Fanuc KAREL source: test_lam.kl

PROGRAM test_lam
%NOLOCKGROUP

%include lam.klt

%include default_lam.klt

VAR
  --work parameters
  lsrprm : t_LASER
  powprm : t_POWDER

%include display.klh
%include lamlib.klh

--lam object
%class tstlam('lam.klc','lam.klh','default_lam.klt')

BEGIN
  --clear display
  display__clear
  --show display
  display__show

  -- --initialize
  -- tstlam__new
  -- tstlam__set_laser_power(3000)
  -- tstlam__set_powder_params(2, POWDER_INCONEL, 2.6, 4, 0.95, 1.27)

  --alternative initalize
  lsrprm = lamlib__new_laser_params(3000)
  powprm = lamlib__new_powder_params(2, POWDER_INCONEL, 2.6, 4, 0.95, 1.27)
  tstlam__init(lsrprm, 2, powprm, FALSE)

  tstlam__set_registers

  WRITE TPDISPLAY('depth: 0.60; speed: ', tstlam__getSpeedFromDepth((powprm.powder), 0.60)::5::2, CR)
  WRITE TPDISPLAY('depth: 1; speed: ', tstlam__getSpeedFromDepth((powprm.powder), 1)::5::2, CR)
  WRITE TPDISPLAY('depth: 1.4; speed: ', tstlam__getSpeedFromDepth((powprm.powder), 1.4)::5::2, CR)

  tstlam__delete

END test_lam
